# EPICS substitutions: si_ps_conv_fastcorrsApp/Db/dipole.substitutions
file "kicks.db"
{
    pattern { DIP, ORI }
            { M1,  FCH }
            { M1,  FCV }
            { M2,  FCH }
            { M2,  FCV }
            { C2,  FCH }
            { C2,  FCV }
            { C3,  FCH }
            { C3,  FCV }
}
